{attribute 'GeneratedUsingTerminal: EK1100-0000-0018'}
{attribute addProperty BoxType "EK1100-0000-0018"}
{attribute addProperty Id "Beckhoff_ELM9xxxEK1122Beckhoff_ELM9xxxEK1122_2662DE952A_0002_ELM9410_0000_0016ELM9410_1354D14381A_0003_ELM9410_0000_0017ELM9410_1354D14381A_0004_ELM9410_0000_0018ELM9410_1354D14381A_0005_ELM9410_0000_0019ELM9410_1354D14381A_0006_ELM9410_0000_0020ELM9410_1354D14381"}
{attribute addProperty CRC "3785044918"}
{attribute addProperty Size "407"}
TYPE Beckhoff_ELM9xxx_E19B33B6 EXTENDS EK1100_AB5A9467 :
STRUCT
	{attribute addProperty Name "Beckhoff_ELM9xxxEK1122"}
	{attribute addProperty PreviousPort "Beckhoff ELM9xxx : B"}
	Beckhoff_ELM9xxxEK1122 : Beckhoff_ELM9xxxEK1122_2662DE95;
	{attribute addProperty Name "A_0002_ELM9410_0000_0016"}
	{attribute addProperty PreviousPort "Beckhoff ELM9xxxEK1122 : C"}
	A_0002_ELM9410_0000_0016 : ELM9410_1354D143;
	{attribute addProperty Name "A_0003_ELM9410_0000_0017"}
	{attribute addProperty PreviousPort "A_0002(ELM9410-0000-0016) : B"}
	A_0003_ELM9410_0000_0017 : ELM9410_1354D143;
	{attribute addProperty Name "A_0004_ELM9410_0000_0018"}
	{attribute addProperty PreviousPort "A_0003(ELM9410-0000-0017) : B"}
	A_0004_ELM9410_0000_0018 : ELM9410_1354D143;
	{attribute addProperty Name "A_0005_ELM9410_0000_0019"}
	{attribute addProperty PreviousPort "A_0004(ELM9410-0000-0018) : B"}
	A_0005_ELM9410_0000_0019 : ELM9410_1354D143;
	{attribute addProperty Name "A_0006_ELM9410_0000_0020"}
	{attribute addProperty PreviousPort "A_0005(ELM9410-0000-0019) : B"}
	A_0006_ELM9410_0000_0020 : ELM9410_1354D143;
END_STRUCT
END_TYPE

(* stored: Version 1.2.0.0, ProductVersion 3.1.4024.9
   DUT Beckhoff_ELM9xxx_E19B33B6: Id {f100b76e-fc2c-48c5-9d77-6aebc9a0c816} *)
